FUNCTION INTERNAL _ArePaired : BOOL
VAR_INPUT
	iSignal				: I_SignalNode;
    iReceiver			: I_ReceiverNode;
END_VAR
VAR_OUTPUT
	nPos				: UDINT;
END_VAR
VAR
	i					: UDINT;
	_nEnd				: UDINT;
END_VAR

IF iSignal.count = 0 THEN
	_ArePaired := FALSE;
	RETURN;	
END_IF

_nEnd := iSignal.id + iSignal.count - 1;
FOR i := iSignal.id TO _nEnd DO
	IF _Channel.stEntry[i].iReceiver = iReceiver THEN
		_ArePaired := TRUE;
		nPos := i;
		RETURN;
	END_IF
END_FOR

END_FUNCTION

(* stored: Version 1.1.0.1
   POU _ArePaired: Id {96f99b54-87d1-48c5-a36c-ed930e76eb5f}, SpecialFunc None *)
